PROGRAM MAIN
VAR
	fbVesselSim: FB_FILL_SIM;
	fbPIControl: FB_CTRL_PI;
	stParameters: ST_CTRL_PI_PARAMS;
	gVessel: TYP_VESSEL;
	bChangeDefaultPi: BOOL;
END_VAR

IF NOT bChangeDefaultPi THEN
	stParameters.bARWOnIPartOnly:=FALSE;
	stParameters.fKp:=200; 
	stParameters.fOutMaxLimit:=100; 
	stParameters.fOutMinLimit:=0; 
	stParameters.tCtrlCycleTime:=T#100MS;
	stParameters.tTaskCycleTime:=T#100MS; 
	stParameters.tTn:=T#2M;
END_IF

fbVesselSim(rFillingRate:=gVessel.rFillingRate, 
			rVesselSize:=gVessel.rVesselSize, 
			rValveInOpening:=fbPIControl.fOut, 
			rEmptyingRate:=gVessel.rEmptyingRate, 
			rValveOutOpening:=gVessel.rValveOutOpening, 
			bReset:=gVessel.bReset);

fbPIControl(fSetpointValue:=gVessel.rSetPoint,
			fActualValue:=fbVesselSim.rVesselLevel,
			eMode:=2,
			fManSyncValue := 50,
			bSync:=FALSE,
			bHold:=FALSE,
			stParams:=stParameters);

END_PROGRAM

(* stored: Version 1.1.0.1, ProductVersion 3.1.4024.12
   POU MAIN: Id {5b0cee5d-8936-4015-a5dc-b49173cf859a}, SpecialFunc None *)
